// TIA Portal V16 export
// export: Created 2022-11-01T21:54:08.9289872Z, ExportSetting WithDefaults, DisplayName Totally Integrated Automation Portal, DisplayVersion V16, DisplayName TIA Portal Version Control Interface, DisplayVersion V16, DisplayName TIA Portal Openness, DisplayVersion V16, DisplayName SINAMICS Startdrive Advanced, DisplayVersion V16, DisplayName SINAMICS Startdrive G130, G150, S120, S150, SINAMICS MV, S210, DisplayVersion V16, DisplayName SINAMICS Startdrive G110M, G120, G120C, G120D, G120P, DisplayVersion V16, DisplayName STEP 7 Professional, DisplayVersion V16, DisplayName STEP 7 Safety, DisplayVersion V16, DisplayName WinCC Professional, DisplayVersion V16
VAR_GLOBAL   // PLC tag table "AI C600"
   iTIR601 AT %MW100 : Int;   // Температура сырья в Е-601
   iTIR602 AT %MW102 : Int;   // Температура сырья перед И-601, после Т-602
   iTIR603 AT %MW104 : Int;   // Температура сырья после И-601 в К-601
   iTIR604 AT %MW106 : Int;   // Температура верха К-601
   iTIR605 AT %MW108 : Int;   // Температура зоны питания К-601
   iTIR606 AT %MW110 : Int;   // Температура низа К-601
   iTIR607 AT %MW112 : Int;   // Температура стабильного бензина с куба К-601 в мтр. Т-602
   iTIR608 AT %MW114 : Int;   // Температура ГЖС после ВХ-601/1,2 в Х-601/1,2
   iTIR609 AT %MW116 : Int;   // Температура ГЖС после Х-601/1,2 в С-601
   iTIR610 AT %MW118 : Int;   // Температура стабильного бензина на ТСБ
   iTIR611 AT %MW120 : Int;   // Температура дымовых газов на выходе из печи П-601 в общую камеру конвекции КУ-601
   iTIR612 AT %MW122 : Int;   // Температура дымовых газов в конвективной части П-601
   iTIR613 AT %MW124 : Int;   // Температура горячей струи на выходе из камеры конвекции в камеру радиации П-601 1-й поток
   iTIR614 AT %MW126 : Int;   // Температура горячей струи на выходе из камеры конвекции в камеру радиации П-601 2-й поток
   iTIR615 AT %MW128 : Int;   // Температура горячей струи на выходе из камеры радиации П-601 1-й поток
   iTIR616 AT %MW130 : Int;   // Температура горячей струи на выходе из камеры радиации П-601 2-й поток
   iTIR617 AT %MW132 : Int;   // Температура горячей струи в куб К-601
   iTIR618 AT %MW134 : Int;   // Температура в Е-602
   iTIR620 AT %MW138 : Int;   // Температура газосырьевой смеси в П-602 после Т-606
   iTIR621 AT %MW140 : Int;   // Температура газопродуктовой смеси перед Т-606
   iTIR623 AT %MW144 : Int;   // Температура газопродуктовой после ВХ-603/1, 2 смеси на входе в сепаратор С-603
   iTIR624 AT %MW146 : Int;   // Температура дымовых газов после П-602 на общую камеру конвекции КУ-601
   iTIR625 AT %MW148 : Int;   // Температура в конвективной части П-602
   iTIR626 AT %MW150 : Int;   // Температура газосырьевой смеси после камеры конвекции в камеру радиации П-602 1-й поток
   iTIR627 AT %MW152 : Int;   // Температура газосырьевой смеси после камеры конвекции в камеру радиации П-602 2-й поток
   iTIR628 AT %MW154 : Int;   // Температура газосырьевой смеси после камеры конвекции в камеру радиации П-602 3-й поток
   iTIR629 AT %MW156 : Int;   // Температура газосырьевой смеси после камеры конвекции в камеру радиации П-602 4-й поток
   iTIR630 AT %MW158 : Int;   // Температура газосырьевой смеси после камеры радиации П-602 1-й поток
   iTIR633 AT %MW164 : Int;   // Температура в Р-601
   iTIR634 AT %MW166 : Int;   // Температура в Р-601
   iTIR635 AT %MW168 : Int;   // Температура в Р-601
   iTIR637 AT %MW172 : Int;   // Температура в Р-601
   iTIR638 AT %MW174 : Int;   // Температура в Р-601
   iTIR639 AT %MW176 : Int;   // Температура газопродуктовой смеси на выходе из Р-601
   iTIR641 AT %MW180 : Int;   // Температура горячей струи в куб К-602 после И-602/2
   iTIR642 AT %MW182 : Int;   // Газопродуктовая смесь в Т-612
   iTIR643 AT %MW184 : Int;   // Температура топливного газа на блок
   iTIR644 AT %MW186 : Int;   // Температура нестабильного ГО бензина в И-602
   iTIR645 AT %MW188 : Int;   // Температура нестабильного ГО бензина после И-602
   iTIR646 AT %MW190 : Int;   // Температура перед ВХ-602/1-3 с верха К-602
   iTIR647 AT %MW192 : Int;   // Температура верха К-602
   iTIR649 AT %MW196 : Int;   // Температура низа К-602
   iTIR650 AT %MW198 : Int;   // Температура тяжелого бензина с низа К-602 в Т-608
   iTIR651 AT %MW200 : Int;   // Температура после ВХ-602/1-3 в С-602
   iTIR652 AT %MW202 : Int;   // Температура после Т-607 к ВХ-602/4
   iTIR653 AT %MW204 : Int;   // Температура после ВХ-602/4
   iTIR654 AT %MW206 : Int;   // Температура обратной воды обратной к Г-601
   iTIR655 AT %MW208 : Int;   // Температура обратной воды подачи после Г-601 на H-5,H-6
   iTIR656_modbus AT %MW210 : Int;   // Температура масла на ПК-603/1
   iPIR601 AT %MW220 : Int;   // Давление на нагнетании Н-601/1,2
   iPIR602 AT %MW222 : Int;   // Давление азотной подушки в Е-601
   iPIR603 AT %MW224 : Int;   // Давление в К-601
   iPIR604 AT %MW226 : Int;   // Давление в С-601, линия УВГ на установку УУФГ
   iPIR605 AT %MW228 : Int;   // Давление горячей струи с нагнетания Н-601/6,7 в П-601
   iPIR606 AT %MW230 : Int;   // Разрежение в П-601
   iPIR607 AT %MW232 : Int;   // Давление топливного газа на форсунки в П-601
   iPIR608 AT %MW234 : Int;   // Давление воздуха на горелки П-601 и П-602
   iPIR609 AT %MW236 : Int;   // Давление азотной подушки в Е-602
   iPIR610 AT %MW238 : Int;   // Давление сырья от Н-602/1,2 в тройник смешения ГО
   iPIR611 AT %MW240 : Int;   // Давление ВСГ на нагнетании компрессора ПК-603/1, 2, 3
   iPIR612 AT %MW242 : Int;   // Давление в сепараторе С-603
   iPIR613 AT %MW244 : Int;   // Давление газосырьевой смеси на входе в П-602
   iPIR614 AT %MW246 : Int;   // Разрежение в П-602
   iPIR617 AT %MW252 : Int;   // Давление после Р-601
   iPIR618 AT %MW254 : Int;   // Давление в К-602
   iPIR619 AT %MW256 : Int;   // Давление в С-602
   iPIR620_virtual AT %MW258 : Int;   // Перепад давления в Р-601
   iPIR621 AT %MW260 : Int;   // Давление в линии топливного газа на блок
   iLIR601 AT %MW300 : Int;   // Уровень в Е-601
   iLIR602 AT %MW302 : Int;   // Уровень в Е-601
   iLIR603 AT %MW304 : Int;   // Уровень в И-601
   iLIR604 AT %MW306 : Int;   // Уровень в кубе К-601
   iLIR605 AT %MW308 : Int;   // Уровень в кубе К-601
   iLIR606 AT %MW310 : Int;   // Уровень сжиженного газа в С-601
   iLIR607 AT %MW312 : Int;   // Уровень сжиженного газа в С-601
   iLIR608 AT %MW314 : Int;   // Уровень кислой воды в С-601
   iLIR609 AT %MW316 : Int;   // Уровень в Е-602
   iLIR610 AT %MW318 : Int;   // Уровень в Е-602
   iLIR611 AT %MW320 : Int;   // Уровень в С-603/1
   iLIR612 AT %MW322 : Int;   // Уровень в С-603/1
   iLIR613 AT %MW324 : Int;   // Уровень нестабильного гидрогенизата в С-603
   iLIR614 AT %MW326 : Int;   // Уровень нестабильного гидрогенизата в С-603
   iLIR615 AT %MW328 : Int;   // Уровень кислой воды в С-603
   iLIR616 AT %MW330 : Int;   // Уровень конденсата в И-602
   iLIR617 AT %MW332 : Int;   // Уровень в К-602
   iLIR618 AT %MW334 : Int;   // Уровень в К-602
   iLIR619 AT %MW336 : Int;   // Уровень в сепараторе С-602
   iLIR620 AT %MW338 : Int;   // Уровень в сепараторе С-602
   iLIR621 AT %MW340 : Int;   // Уровень кислой воды в сепараторе С-602
   iLIR622 AT %MW342 : Int;   // Уровень в факельном сепараторе С-607
   iLIR623 AT %MW344 : Int;   // Уровень кислой воды в Е-905/1
   iLIR624 AT %MW346 : Int;   // Уровень кислой воды в Е-905/2
   iLIR625 AT %MW348 : Int;   // Уровень кислой воды в Е-607
   iFIR601 AT %MW420 : Int;   // Расход КГЛУ с ТСБ, конденсата с УУФГ от С-403/2 на установку получения сжиженного газа
   iFIR602 AT %MW422 : Int;   // Расход сырья К-601 от Н-601/1,2 в Т-601
   iFIR603 AT %MW424 : Int;   // Расход топливного газа на блок
   iFIR604 AT %MW426 : Int;   // Расход пароконденсата после И-601
   iFIR605 AT %MW428 : Int;   // Расход орошения в К-601
   iFIR606 AT %MW430 : Int;   // Расход сжиженного газа из сепаратора С-601 на ТСБ
   iFIR607 AT %MW432 : Int;   // Расход УВГ из сепаратора С-601 на УУФГ
   iFIR608 AT %MW434 : Int;   // Расход стабильного бензина из К-601 на ТСБ
   iFIR609 AT %MW436 : Int;   // Расход горячей струи в П-601 от Н-601/6,7
   iFIR610 AT %MW438 : Int;   // Расход горячей струи в П-601 1-й поток
   iFIR611 AT %MW440 : Int;   // Расход горячей струи в П-601 2-й поток
   iFIR612 AT %MW442 : Int;   // Расход циркуляции сырья с нагнетания Н-602/1,2 в Е-602
   iFIR613 AT %MW444 : Int;   // Расход сырья от Н-602/1,2 в тройник смешения гидроочистки
   iFIR614 AT %MW446 : Int;   // Расход сырья от Н-602/1,2 в тройник смешения гидроочистки
   iFIR615 AT %MW448 : Int;   // Расход ВСГ от ПК-603/1-3 в тройник смешения гидроочистки
   iFIR616 AT %MW450 : Int;   // Расход ВСГ от ПК-603/1-3 в тройник смешения гидроочистки
   iFIR617 AT %MW452 : Int;   // Расход подпиточного ВСГ в приемный сепаратор С-603/1 циркуляционного компрессора ПК-603/1-3
   iFIR618 AT %MW454 : Int;   // Расход нестабильного гидрогенизата из С-603 в Т-607
   iFIR619 AT %MW456 : Int;   // Расход сдувки ВСГ из С-603 в Е-903
   iFIR620 AT %MW458 : Int;   // Расход пароконденсата после И-602
   iFIR621 AT %MW460 : Int;   // Расход орошения в К-602
   iFIR622 AT %MW462 : Int;   // Расход УВГ из С-602 в Е-903
   iFIR623 AT %MW464 : Int;   // Расход дистиллята К-602 в Е-501
   iFIR624 AT %MW466 : Int;   // Расход стабильного ГО бензина на ТСБ или в Е-603
   iFIR625 AT %MW468 : Int;   // Расход оборотной воды от Н-615/1,2
   iTIR619 AT %MW136 : Int;   // Температура ВСГ после ПК-603/1, 2, 3 в тройник смешения ГО
   iTIR622 AT %MW142 : Int;   // Температура газопродуктовой смеси после Т-603 перед ВХ-603/1, 2
   iTIR631 AT %MW160 : Int;   // Температура газосырьевой смеси после камеры радиации П-602 2-й поток
   iTIR632 AT %MW162 : Int;   // Температура газосырьевой смеси после П-602 в Р-601
   iTIR640 AT %MW178 : Int;   // Температура горячей струи в куб К-602 после И-602/1
   iTIR648 AT %MW194 : Int;   // Температура зоны питания К-602
   iTIR657_modbus AT %MW212 : Int;   // Температура масла на ПК-603/2
   iTIR658_modbus AT %MW214 : Int;   // Температура масла на ПК-603/3
   iTIR636 AT %MW170 : Int;   // Температура в Р-601
   iPIR615 AT %MW248 : Int;   // Давление топливного газа на форсунки в П-602
   iPIR616 AT %MW250 : Int;   // Давления на входе в Р-601
   iPIR622_modbus AT %MW262 : Int;   // Давление ВСГ на всасе компрессора ПК-603/1
   iPIR623_modbus AT %MW264 : Int;   // Давление ВСГ на нагнетании компрессора ПК-603/1
   iPIR624_modbus AT %MW266 : Int;   // Давление масла на компрессоре ПК-603/1
   iPIR625_modbus AT %MW268 : Int;   // Давление ВСГ на всасе компрессора ПК-603/2
   iPIR626_modbus AT %MW270 : Int;   // Давление ВСГ на нагнетании компрессора ПК-603/2
   iPIR627_modbus AT %MW272 : Int;   // Давление масла на компрессоре ПК-603/2
   iPIR628_modbus AT %MW274 : Int;   // Давление ВСГ на всасе компрессора ПК-603/3
   iPIR629_modbus AT %MW276 : Int;   // Давление ВСГ на нагнетании компрессора ПК-603/3
   iPIR630_modbus AT %MW278 : Int;   // Давление масла на компрессоре ПК-603/3
   iQIR601 AT %MW216 : Int;   // Содержание кислорода в дымовых газах печи П-601
   iQIR602 AT %MW218 : Int;   // Содержание кислорода в дымовых газах печи П-602
END_VAR
